(* IEC 61131-3 sources: AXOpen/src/core/ctrl/src/abstractions, 6 files *)

(* ---- IAxoLogger.st ---- *)
USING AXOpen.Core;
USING AXOpen.Core;
NAMESPACE AXOpen.Messaging

    TYPE
        eLogLevel : INT (NoCat := 0, Verbose := 1, Debug  := 2, Information  := 3, Warning  := 4, Error  := 5, Fatal  := 6) := NoCat;
    END_TYPE

    INTERFACE PUBLIC IAxoLogger
        METHOD Log
            VAR_INPUT
                _message : STRING[80];
                _level : eLogLevel;
                _sender : IAxoObject;
            END_VAR
        END_METHOD
    END_INTERFACE

    INTERFACE IAxoLoggerConfig
        METHOD MinimumLevel : IAxoLoggerConfig
            VAR_INPUT
                _level : eLogLevel;
            END_VAR
        END_METHOD
    END_INTERFACE
END_NAMESPACE

(* ---- IContext.st ---- *)
NAMESPACE ix.framework.core
    INTERFACE IContext
        METHOD CreateIdentity : ULINT END_METHOD
        METHOD OpenCycleCount : ULINT END_METHOD
    END_INTERFACE
END_NAMESPACE

(* ---- IIxContext.st ---- *)
NAMESPACE ix.framework.core
    INTERFACE IIxContext
        METHOD CreateIdentity : ULINT END_METHOD
        METHOD OpenCycleCount : ULINT END_METHOD
    END_INTERFACE
END_NAMESPACE

(* ---- IIxObject.st ---- *)
NAMESPACE ix.framework.core
  INTERFACE IIxObject
    METHOD GetIdentity : ULINT  END_METHOD
    METHOD GetContext : IIxContext END_METHOD
  END_INTERFACE
END_NAMESPACE

(* ---- IObject.st ---- *)
NAMESPACE ix.framework.core
  INTERFACE IObject
    METHOD GetIdentity : ULINT  END_METHOD
    METHOD GetContext : IContext END_METHOD
  END_INTERFACE
END_NAMESPACE

(* ---- NULLs.st ---- *)
USING AXOpen.Messaging;
USING AXOpen.Logging;
USING AXOpen.Rtc;
USING AXOpen.Rtm;

NAMESPACE AXOpen.Core
    ///<summary>
    /// Provides an empty context for uninitialized objects.
    ///</summary>
    CLASS PUBLIC _NULL_CONTEXT IMPLEMENTS IAxoContext
        VAR PRIVATE
            {S7.extern=Hidden}
            NULL_RTC : _NULL_RTC;
            {S7.extern=Hidden}
            NULL_LOGGER : _NULL_LOGGER;
            {S7.extern=Hidden}
            NULL_RTM : _NULL_RTM;
        END_VAR

        METHOD PUBLIC CreateIdentity : ULINT CreateIdentity := ULINT#0; END_METHOD
        METHOD PUBLIC OpenCycleCount : ULINT OpenCycleCount := ULINT#0; END_METHOD
        METHOD PUBLIC GetRtc : IAxoRtc GetRtc := NULL_RTC; END_METHOD
        METHOD PUBLIC InjectRtc VAR_INPUT Rtc : IAxoRtc; END_VAR ; END_METHOD
        METHOD PUBLIC GetLogger : IAxoLogger GetLogger :=  NULL_LOGGER; END_METHOD
        METHOD PUBLIC InjectLogger VAR_INPUT _logger : IAxoLogger; END_VAR ; END_METHOD
        METHOD PUBLIC GetRtm : IAxoRtm GetRtm :=  NULL_RTM; END_METHOD
        METHOD PUBLIC InjectRtm VAR_INPUT rtm : IAxoRtm; END_VAR ; END_METHOD

    END_CLASS

    ///<summary>
    /// Provides an empty object for uninitialized objects.
    ///</summary>
    CLASS PUBLIC _NULL_OBJECT IMPLEMENTS IAxoObject
        VAR PRIVATE
            {S7.extern=Hidden}
            NULL_CONTEXT : _NULL_CONTEXT;
        END_VAR
        METHOD PUBLIC GetIdentity : ULINT
            GetIdentity := ULINT#0;
        END_METHOD
        METHOD PUBLIC GetContext : IAxoContext
            GetContext := NULL_CONTEXT;
        END_METHOD
        METHOD PUBLIC GetContextUnsafe : IAxoContext
            GetContextUnsafe := NULL_CONTEXT;
    END_METHOD
    END_CLASS

    ///<summary>
    /// Provides an empty RTC object for uninitialized RTC.
    ///</summary>
    {S7.extern=ReadWrite}
    CLASS PUBLIC _NULL_RTC IMPLEMENTS IAxoRtc
        VAR PRIVATE
            _null_time : LDATE_AND_TIME := LDATE_AND_TIME#1970-01-01-00:00:00.000;
        END_VAR
        METHOD PUBLIC NowUTC : LDATE_AND_TIME
            NowUTC := _null_time;
        END_METHOD
    END_CLASS

    ///<summary>
    /// Provides an empty logger object for uninitialized context logger.
    ///</summary>
    {S7.extern=ReadWrite}
    CLASS PUBLIC _NULL_LOGGER IMPLEMENTS IAxoLogger
        METHOD PUBLIC Log
            VAR_INPUT
                _message : STRING[80];
                _level : eLogLevel;
                _sender : IAxoObject;
            END_VAR
            ;
        END_METHOD

        METHOD PUBLIC Log
            VAR_INPUT
                _message : STRING[80];
                _level : eLogLevel;
            END_VAR
            ;
        END_METHOD

        METHOD PUBLIC SetMinimumLevel : IAxoLoggerConfig
            VAR_INPUT
                _level : eLogLevel;
            END_VAR
            ;
        END_METHOD
    END_CLASS

    ///<summary>
    /// Provides an empty RTC object for uninitialized RTC.
    ///</summary>
    {S7.extern=ReadWrite}
    CLASS PUBLIC _NULL_RTM IMPLEMENTS IAxoRtm
        VAR PRIVATE
            _null_time : LTIME;
        END_VAR

        METHOD PUBLIC Elapsed : LTIME
            Elapsed := _null_time;
        END_METHOD
    END_CLASS
END_NAMESPACE
